(* CoDeSys 2.3.9.48 project: XV400_Profibus_XNE2cntComptage simple.pro *)
(* Libraries: Standard.lib 5.4.06 13:34:00, Util.lib 20.3.15 09:30:08, SysLibCallback.lib 21.5.10 07:41:54, SysLibSockets.lib 7.5.14 07:02:16, SysLibTasks.lib 3.7.08 07:33:54, SysLibRtc.lib 29.9.06 14:48:48, SysLibFile.lib 29.9.06 14:48:48, SysLibPlcCtrl.lib 29.9.06 14:48:48, 3S_CanDrv.lib 27.3.12 16:31:06, 3S_CANopenManager.lib 30.3.15 10:04:38, 3S_CANopenMaster.lib 27.3.15 07:15:26, CanUser.lib 27.3.12 16:31:06, CanUser_Master.lib 28.4.15 13:38:54, SysLibForce.lib 3.7.08 07:33:54 *)

(* Global variable list: CanOpen implicit Variables *)
VAR_GLOBAL CONSTANT
	MAX_CTRLINDEX : INT := 0;
END_VAR
VAR_GLOBAL CONSTANT
	USE_CANOPEN_NODES : BOOL := FALSE;
	MAX_MASTERINDEX : INT := 0;
	MAX_NODEINDEX : INT := 0;
	MAX_SDOINDEX : INT := 0;
	MAX_PDOINDEX_RX : INT := 0;
	MAX_PDOINDEX_TX : INT := 0;
END_VAR
VAR_GLOBAL
	pCANopenMaster : ARRAY[0..MAX_MASTERINDEX] OF CanOpenMaster;
	pCanOpenNode : ARRAY[0..MAX_NODEINDEX] OF CanOpenNode;
	pCanOpenSDO : ARRAY[0..MAX_SDOINDEX] OF CanOpenSDO;
	pCanOpenPDO_Rx : ARRAY[0..MAX_PDOINDEX_RX] OF CanOpenPDO_Rx;
	pCanOpenPDO_Tx : ARRAY[0..MAX_PDOINDEX_TX] OF CanOpenPDO_Tx;
END_VAR

(* POU PLC_PRG, ST *)
PROGRAM PLC_PRG
VAR
	Control_A1: BYTE;
END_VAR
%QB0 := Control_A1; (* forcer avec la page de visu *)

%IB0;
%IB1;
%IB2;
%IB3;
%IB4;
%IB5;
%IB6;
%IB7;
%IB8;
%IB9;
%IB10;
%IB11;
%IB12;
%IB13;
%IB14;
%IB15;
END_PROGRAM

(* Visualisation MAPAGE
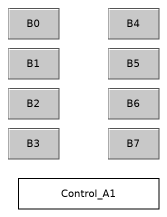
button at (10,10)-(61,41): text "B0"; toggles PLC_PRG.Control_A1.0
button at (110,10)-(161,41): text "B4"; toggles PLC_PRG.Control_A1.4
button at (10,50)-(61,81): text "B1"; toggles PLC_PRG.Control_A1.1
button at (10,90)-(61,121): text "B2"; toggles PLC_PRG.Control_A1.2
button at (10,130)-(61,161): text "B3"; toggles PLC_PRG.Control_A1.3
button at (110,50)-(161,81): text "B5"; toggles PLC_PRG.Control_A1.5
button at (110,90)-(161,121): text "B6"; toggles PLC_PRG.Control_A1.6
button at (110,130)-(161,161): text "B7"; toggles PLC_PRG.Control_A1.7
rectangle at (20,180)-(161,211): text "Control_A1"
*)
